// TIA Portal V16 export
// export: Created 2023-03-29T11:04:46.8690165Z, ExportSetting WithDefaults, DisplayName Totally Integrated Automation Portal, DisplayVersion V16 Update 6, DisplayName TIA Portal Version Control Interface, DisplayVersion V16 Update 2, DisplayName TIA Portal Openness, DisplayVersion V16 Update 6, DisplayName STEP 7 Professional, DisplayVersion V16 Update 6, DisplayName STEP 7 Safety, DisplayVersion V16, DisplayName WinCC Advanced, DisplayVersion V16 Update 6
FUNCTION "Blok liczników pracy" : Void   // FC8, LAD
TITLE = Wywołanie funkcji liczników pracy
{ S7_Optimized_Access := 'TRUE' }
AUTHOR : RTecmer
VERSION : 0.1
// Funkcja wywołuje liczniki pracy napędów
// stored: AutoNumber true, IsIECCheckEnabled false, SetENOAutomatically false, UDAEnableTagReadback false
BEGIN

REGION Network 1: Pompa P1
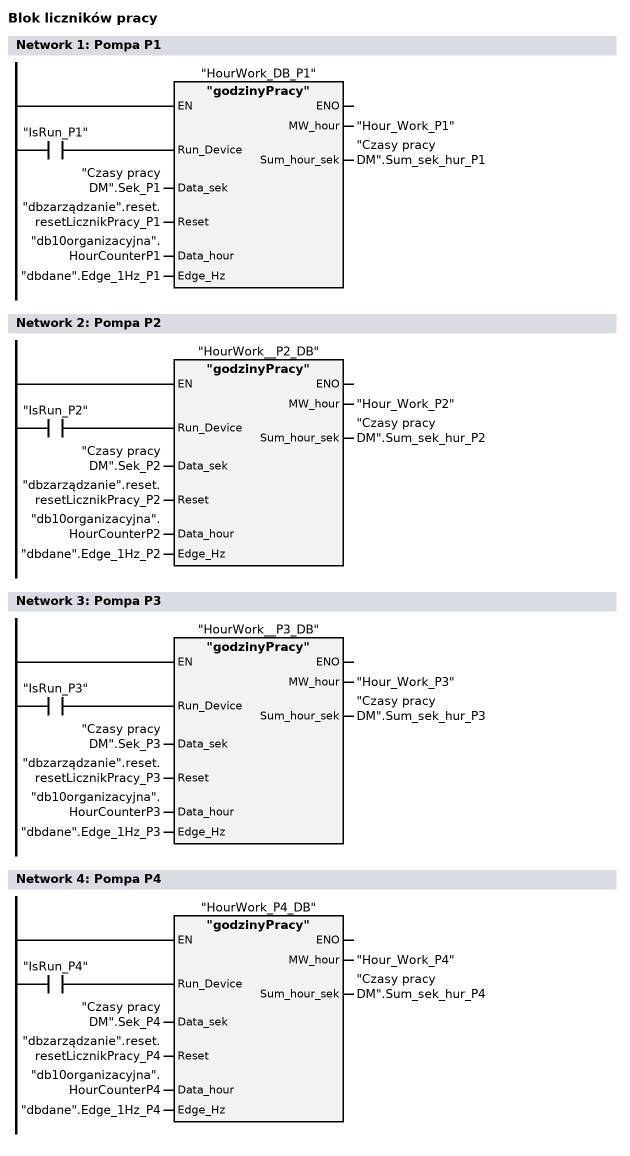
   RUNG wire#powerrail
      "HourWork_DB_P1"(Run_Device := wire#w1, Data_sek := "Czasy pracy DM".Sek_P1, Reset := "dbzarządzanie".reset.resetLicznikPracy_P1, Data_hour := "db10organizacyjna".HourCounterP1, Edge_Hz := "dbdane".Edge_1Hz_P1, MW_hour => "Hour_Work_P1", Sum_hour_sek => "Czasy pracy DM".Sum_sek_hur_P1)
   END_RUNG
   RUNG wire#powerrail
      Contact( "IsRun_P1" )
   END_RUNG wire#w1
   // the same network as SCL:
   "HourWork_DB_P1"(Run_Device := "IsRun_P1",   // "godzinyPracy"
                    Data_sek := "Czasy pracy DM".Sek_P1,
                    Reset := "dbzarządzanie".reset.resetLicznikPracy_P1,
                    Data_hour := "db10organizacyjna".HourCounterP1,
                    Edge_Hz := "dbdane".Edge_1Hz_P1,
                    MW_hour => "Hour_Work_P1",
                    Sum_hour_sek => "Czasy pracy DM".Sum_sek_hur_P1);
END_REGION

REGION Network 2: Pompa P2
   RUNG wire#powerrail
      "HourWork__P2_DB"(Run_Device := wire#w1, Data_sek := "Czasy pracy DM".Sek_P2, Reset := "dbzarządzanie".reset.resetLicznikPracy_P2, Data_hour := "db10organizacyjna".HourCounterP2, Edge_Hz := "dbdane".Edge_1Hz_P2, MW_hour => "Hour_Work_P2", Sum_hour_sek => "Czasy pracy DM".Sum_sek_hur_P2)
   END_RUNG
   RUNG wire#powerrail
      Contact( "IsRun_P2" )
   END_RUNG wire#w1
   // the same network as SCL:
   "HourWork__P2_DB"(Run_Device := "IsRun_P2",   // "godzinyPracy"
                     Data_sek := "Czasy pracy DM".Sek_P2,
                     Reset := "dbzarządzanie".reset.resetLicznikPracy_P2,
                     Data_hour := "db10organizacyjna".HourCounterP2,
                     Edge_Hz := "dbdane".Edge_1Hz_P2,
                     MW_hour => "Hour_Work_P2",
                     Sum_hour_sek => "Czasy pracy DM".Sum_sek_hur_P2);
END_REGION

REGION Network 3: Pompa P3
   RUNG wire#powerrail
      "HourWork__P3_DB"(Run_Device := wire#w1, Data_sek := "Czasy pracy DM".Sek_P3, Reset := "dbzarządzanie".reset.resetLicznikPracy_P3, Data_hour := "db10organizacyjna".HourCounterP3, Edge_Hz := "dbdane".Edge_1Hz_P3, MW_hour => "Hour_Work_P3", Sum_hour_sek => "Czasy pracy DM".Sum_sek_hur_P3)
   END_RUNG
   RUNG wire#powerrail
      Contact( "IsRun_P3" )
   END_RUNG wire#w1
   // the same network as SCL:
   "HourWork__P3_DB"(Run_Device := "IsRun_P3",   // "godzinyPracy"
                     Data_sek := "Czasy pracy DM".Sek_P3,
                     Reset := "dbzarządzanie".reset.resetLicznikPracy_P3,
                     Data_hour := "db10organizacyjna".HourCounterP3,
                     Edge_Hz := "dbdane".Edge_1Hz_P3,
                     MW_hour => "Hour_Work_P3",
                     Sum_hour_sek => "Czasy pracy DM".Sum_sek_hur_P3);
END_REGION

REGION Network 4: Pompa P4
   RUNG wire#powerrail
      "HourWork_P4_DB"(Run_Device := wire#w1, Data_sek := "Czasy pracy DM".Sek_P4, Reset := "dbzarządzanie".reset.resetLicznikPracy_P4, Data_hour := "db10organizacyjna".HourCounterP4, Edge_Hz := "dbdane".Edge_1Hz_P4, MW_hour => "Hour_Work_P4", Sum_hour_sek => "Czasy pracy DM".Sum_sek_hur_P4)
   END_RUNG
   RUNG wire#powerrail
      Contact( "IsRun_P4" )
   END_RUNG wire#w1
   // the same network as SCL:
   "HourWork_P4_DB"(Run_Device := "IsRun_P4",   // "godzinyPracy"
                    Data_sek := "Czasy pracy DM".Sek_P4,
                    Reset := "dbzarządzanie".reset.resetLicznikPracy_P4,
                    Data_hour := "db10organizacyjna".HourCounterP4,
                    Edge_Hz := "dbdane".Edge_1Hz_P4,
                    MW_hour => "Hour_Work_P4",
                    Sum_hour_sek => "Czasy pracy DM".Sum_sek_hur_P4);
END_REGION
END_FUNCTION
